PROGRAM Main
VAR
	PowerOn			: bool	:= true;	// initialize on, turn false on second scan
	FirstRun		: BOOL := TRUE;		// initialize on, turn false when system has reached starting postion 

	i						: UINT;				// loop index variable
	Step					: XTSSequence;		// primary sequencer
	stCaGroupRef			: AXES_GROUP_REF;
	fbEnableGroup			: MC_GroupEnable;
	fbAddAxis				: ARRAY[1..GVL.NUM_MOVERS] OF MC_AddAxisToGroup;
	fbRemoveAxisFromGroup	: ARRAY[1..GVL.NUM_MOVERS] OF MC_RemoveAxisFromGroup;
	nAtStart: UINT;
	nToStart: UINT;
	
	allMoversHalted: BOOL;

	
	
	MoversReady: BOOL;
	Started: BOOL;
	Resumed: BOOL;
	bLightCurtainEntered: R_TRIG;
	bLightCurtainExited: F_TRIG;
END_VAR

(* this program handles the main sequencer of this machine *)

// cyclic call to execute fb's for movers, stations, and zones
FOR i := 1 TO GVL.NUM_MOVERS DO
	GVL.Mover[i]();
	GVL.Mover[i].AxisReference.ReadStatus();
	fbRemoveAxisFromGroup[i](AxesGroup		:= stCaGroupRef);
	fbAddAxis[i](AxesGroup		:= stCaGroupRef,
				Axis			:= GVL.Mover[i].AxisReference);
				
	IF GVL.Mover[i].AxisReference.Status.Moving THEN
				allMoversHalted		:= FALSE;
			END_IF
END_FOR
FOR i := 1 TO GVL.NUM_STATIONS DO
	GVL.Station[i]();
END_FOR
FOR i := 1 TO gvl.NUM_ZONES DO
	GVL.Zone[i]();
END_FOR

// check for HMI STOP/PAUSE
IF HMI.Stop THEN
	HMI.Stop	:= FALSE;
	Step		:= XTSSequence.Stop;
ELSIF HMI.Pause THEN
	HMI.Pause	:= FALSE;
	Step		:= XTSSequence.Pause;
END_IF

CASE Step OF

//-----------------------------------------------------------------------------------------------------------------------	
	XTSSequence.Off:
		// state waiting for start command		----	Movers are off
		
		
		
		//COMMIT TEST
		
		Initialize();

			IF HMI.StartOver THEN
				Step		:= XTSSequence.EnableMovers;
				Started := TRUE;
				HMI.StartOver := FALSE;
			END_IF
			
			IF HMI.Resume THEN
				Step			:= XTSSequence.EnableMovers;
				Resumed := TRUE;
				HMI.Resume := FALSE;
			END_IF

//-----------------------------------------------------------------------------------------------------------------------	
	XTSSequence.Pause:
	
	FOR i := 1 TO GVL.NUM_MOVERS  DO
		GVL.Mover[i].toPause := TRUE;
	END_FOR
	
	Started := FALSE;
	Resumed := FALSE;
	Step := XTSSequence.Pausing;
	
//-----------------------------------------------------------------------------------------------------------------------	
	XTSSequence.Pausing:
	
	// Waiting for all to come to a full stop
	allMoversHalted				:= TRUE;
	
	FOR i := 1 TO GVL.NUM_MOVERS DO
		IF GVL.Mover[i].AxisReference.Status.Moving THEN
			allMoversHalted		:= FALSE;
		END_IF
	END_FOR
	
	IF allMoversHalted THEN
		Step		:= XTSSequence.Off;
	END_IF

//-----------------------------------------------------------------------------------------------------------------------	
	XTSSequence.Stop:
	
	FOR i := 1 TO GVL.NUM_MOVERS  DO
		GVL.Mover[i].toStop := TRUE;
	END_FOR
	
	Started := FALSE;
	Resumed := FALSE;
	Step		:= XTSSequence.Stopping;
		
//-----------------------------------------------------------------------------------------------------------------------	
	XTSSequence.Stopping:
		// Waiting for all to come to a full stop
		allMoversHalted				:= TRUE;
	
		FOR i := 1 TO GVL.NUM_MOVERS DO
			IF GVL.Mover[i].AxisReference.Status.Moving THEN
				allMoversHalted		:= FALSE;
			END_IF
		END_FOR
	
	IF allMoversHalted THEN
		Step		:= XTSSequence.RemoveAxes;
	END_IF
	
//-----------------------------------------------------------------------------------------------------------------------	
	XTSSequence.RemoveAxes:
		// remove all axes to collision avoidance group
		// loop through each mover axis and remove CA group
		FOR i:= 1 TO GVL.NUM_MOVERS DO
			fbRemoveAxisFromGroup[i].IdentInGroup := UDINT_TO_IDENTINGROUP(UINT_TO_UDINT(i));
			fbRemoveAxisFromGroup[i].Execute			:= TRUE;
		END_FOR
	
		IF stCaGroupRef.NcToPlc.CA.Common.GroupAxesCount = 0 THEN
			FOR i:= 1 TO GVL.NUM_MOVERS DO
				fbRemoveAxisFromGroup[i].IdentInGroup	:= UDINT_TO_IDENTINGROUP(UINT_TO_UDINT(i));
				fbRemoveAxisFromGroup[i].Execute			:= FALSE;
				MoversReady := FALSE;
		END_FOR
			Step := XTSSequence.DisableMovers;
		END_IF

//-----------------------------------------------------------------------------------------------------------------------	
	XTSSequence.DisableMovers:
	FOR i := 1 TO GVL.NUM_MOVERS  DO
		GVL.Mover[i].toDisable := TRUE;
	END_FOR
	
	Step := XTSSequence.Off;
		
//-----------------------------------------------------------------------------------------------------------------------			
	XTSSequence.EnableMovers:
		// enable all movers
		FOR i := 1 TO GVL.NUM_MOVERS DO
			IF NOT GVL.Mover[i].Enabled THEN
				GVL.Mover[i].Enable	:= TRUE;
			END_IF
		END_FOR
		
		// check for all enabled
		FOR i := 1 TO GVL.NUM_MOVERS DO
			IF NOT GVL.Mover[i].Enabled THEN
				// not enabled, leave for loop
				EXIT;
			END_IF
			// made it this far, all movers are enabled
			IF i = gvl.NUM_MOVERS THEN
				Step	:= XTSSequence.EnableGroup;
			END_IF
		END_FOR
		
//-----------------------------------------------------------------------------------------------------------------------		
	XTSSequence.EnableGroup:
	// enable CA group
	fbEnableGroup.Execute := TRUE;
	// verify group enabled successfully
	IF fbEnableGroup.Done = TRUE THEN
		fbEnableGroup.Execute := FALSE;
		Step := XTSSequence.AddAxes;
	END_IF
		
//-----------------------------------------------------------------------------------------------------------------------		
	XTSSequence.AddAxes:
		// add all axes to collision avoidance group
		// loop through each mover axis and add to CA group
	FOR i:= 1 TO GVL.NUM_MOVERS DO
		fbAddAxis[i].IdentInGroup := UDINT_TO_IDENTINGROUP(UINT_TO_UDINT(i));
		fbAddAxis[i].Execute := TRUE;
	END_FOR
	
	// verify all axes added
	IF stCaGroupRef.NcToPlc.CA.Common.GroupAxesCount = GVL.NUM_MOVERS THEN
		FOR i:= 1 TO GVL.NUM_MOVERS DO
			fbAddAxis[i].IdentInGroup := UDINT_TO_IDENTINGROUP(UINT_TO_UDINT(i));
			fbAddAxis[i].Execute := FALSE;
			MoversReady := TRUE;
			Step	:= XTSSequence.StandBy;
		END_FOR
	END_IF
		
//-----------------------------------------------------------------------------------------------------------------------		
	XTSSequence.StandBy:
	IF Started THEN
		// first time code executes this far (after power on) move to a start position
		Started := FALSE;
		Step	:= XTSSequence.Start;
	ELSIF Resumed THEN
		// any other time code executes here, resume operation where movers left off
		Resumed := FALSE;
		Step	:= XTSSequence.Run;
	END_IF

//-----------------------------------------------------------------------------------------------------------------------		
	XTSSequence.Start:
		// request all movers proceed to starting station
IF HMI.bzone0Stop = FALSE THEN
	FOR i:= 1 TO GVL.NUM_MOVERS DO
		GVL.Mover[i].toStart	:= TRUE;
	END_FOR
	// verify one mover is at start, all others have commands and are at zero speed
	nAtStart	:= 0;
	nToStart	:= 0;
	FOR i:= 1 TO GVL.NUM_MOVERS DO
		IF GVL.Mover[i].Step = MoverSequence.AtStart THEN
			nAtStart	:= nAtStart + 1;
		ELSIF GVL.Mover[i].Step = MoverSequence.MovingToStart THEN
			nToStart	:= nToStart + 1;
		END_IF
	END_FOR
	IF nAtStart = 1 AND nToStart = GVL.NUM_MOVERS - 1 THEN
		Step	:= XTSSequence.Run;
	END_IF
END_IF	
//-----------------------------------------------------------------------------------------------------------------------	
	XTSSequence.Run:
	(*
	FOR i:= 1 TO GVL.NUM_MOVERS DO
			GVL.Mover[i].toNext	:= TRUE;
		END_FOR
	*)
	
	// LOAD TRAY STATION
	IF GVL.Station[1].Step = StationSequence.MoverPresent THEN
		HMI.dsMoverControlFlags.loadTray_Busy := TRUE;
		IF HMI.dsMoverControlFlags.loadTray_Complete THEN			//IF SENSOR IS TRUE PACKAGE IS PRESENT MOVER GOES TO NEXT STATION
			HMI.dsMoverControlFlags.loadTray_Complete := FALSE;
			GVL.Station[1].bMoveToNext := TRUE;
		END_IF
	ELSE
		HMI.dsMoverControlFlags.loadTray_Busy := FALSE;
	END_IF
	
	// LOAD PARTS STATION 1
	IF GVL.Station[2].Step = StationSequence.MoverPresent THEN
		HMI.dsMoverControlFlags.loadArea1_Busy := TRUE;				//SIGNAL TO ROBOT 1 TO LOAD PARTS
		IF HMI.dsMoverControlFlags.loadArea1_Complete THEN			//SIGNAL FROM ROBOT 1 PARTS COMPLETED
			HMI.dsMoverControlFlags.loadArea1_Complete := FALSE;
			GVL.Station[2].bMoveToNext := TRUE;
		END_IF
	ELSE 
		HMI.dsMoverControlFlags.loadArea1_Busy := FALSE;
	END_IF
	
	// LOAD PARTS STATION 2
	IF GVL.Station[3].Step = StationSequence.MoverPresent THEN
		HMI.dsMoverControlFlags.loadArea2_Busy := TRUE;				//SIGNAL TO ROBOT 2 TO LOAD PARTS
		IF HMI.dsMoverControlFlags.loadArea2_Complete THEN			//SIGNAL FROM ROBOT 2 PARTS COMPLETED
			HMI.dsMoverControlFlags.loadArea2_Complete := FALSE;
			GVL.Station[3].bMoveToNext := TRUE;
		END_IF
	ELSE
		HMI.dsMoverControlFlags.loadArea2_Busy := FALSE;	
	END_IF
	
	// LOAD PARTS STATION 3
	IF GVL.Station[4].Step = StationSequence.MoverPresent THEN
		HMI.dsMoverControlFlags.loadArea3_Busy := TRUE;				//SIGNAL TO ROBOT 3 TO LOAD PARTS
		IF HMI.dsMoverControlFlags.loadArea3_Complete THEN			//SIGNAL FROM ROBOT 3 PARTS COMPLETED
			HMI.dsMoverControlFlags.loadArea3_Complete := FALSE;
			GVL.Station[4].bMoveToNext := TRUE;
		END_IF
	ELSE
		HMI.dsMoverControlFlags.loadArea3_Busy := FALSE;
	END_IF

	// LOAD PARTS STATION 4
	IF GVL.Station[5].Step = StationSequence.MoverPresent THEN
		HMI.dsMoverControlFlags.loadArea4_Busy := TRUE;				//SIGNAL TO ROBOT 4 TO LOAD PARTS
		IF HMI.dsMoverControlFlags.loadArea4_Complete THEN			//SIGNAL FROM ROBOT 4 PARTS COMPLETED
			HMI.dsMoverControlFlags.loadArea4_Complete := FALSE;
			GVL.Station[5].bMoveToNext := TRUE;
		END_IF
	ELSE
		HMI.dsMoverControlFlags.loadArea4_Busy := FALSE;	
	END_IF
	
	// UNLOAD PARTS STATION 
	IF GVL.Station[6].Step = StationSequence.MoverPresent THEN
		HMI.dsMoverControlFlags.unloadTray_Busy := TRUE;			//SIGNAL TO ROBOT 5 TO UNLOAD TRAY
		IF HMI.dsMoverControlFlags.unloadTray_Complete THEN			//SIGNAL FROM ROBOT 5 UNLOAD TRAY COMPLETED
			HMI.dsMoverControlFlags.unloadTray_Complete := FALSE;
			IF HMI.bzone0Stop THEN
				GVL.Station[6].bMoveToNext := TRUE;					//Send to Queue Movers Station
			ELSE
				GVL.Station[6].bMoveToStart := TRUE;					//Send to Load Tray Station
			END_IF

		END_IF
	ELSE
		HMI.dsMoverControlFlags.unloadTray_Busy := FALSE;
	END_IF
	
	// Queue Station used only if Operator is in Zone 1
	IF GVL.Station[7].Step = StationSequence.MoverPresent THEN
		IF HMI.bzone0Stop = FALSE THEN			
			GVL.Station[7].bMoveToStart := TRUE;
		END_IF
	END_IF
	
	IF HMI.StartOver THEN
		Started := TRUE;
		HMI.StartOver := FALSE;
		Step :=	XTSSequence.Standby;
		
	END_IF
	
END_CASE

fbEnableGroup(AxesGroup	:= stCaGroupRef);
LightCurtainCheck();

METHOD Initialize : BOOL
VAR_INPUT
END_VAR
// set values of function blocks
	GVL.Station[1].Position		:= 0.0;
	GVL.Station[2].Position		:= 750.0;
	GVL.Station[3].Position		:= 1500.0;
	GVL.Station[4].Position		:= 2250.0;
	GVL.Station[5].Position		:= 3000.0;
	GVL.Station[6].Position		:= 3600.0;
	GVL.Station[7].Position		:= 4250.0;
	GVL.Station[8].Position		:= 4490.0;
END_METHOD

ACTION LightCurtainCheck:
// ZONE 0  OPERATER LOADING
bLightCurtainEntered(CLK:=HMI.bzone0Stop);
bLightCurtainExited(CLK:=HMI.bzone0Stop);
	IF bLightCurtainEntered.Q THEN
		FOR i:= 1 TO GVL.NUM_MOVERS DO	
			IF GVL.Mover[i].Position >= 4500.0 OR GVL.Mover[i].Position <= 500.0 THEN
			GVL.Mover[i].toPause	:= TRUE;
			GVL.Mover[i].toNext		:= FALSE;
			GVL.Mover[i].toStart	:= FALSE;
			END_IF
		END_FOR
	END_IF
	IF bLightCurtainExited.Q THEN
		FOR i:= 1 TO GVL.NUM_MOVERS DO	
			IF GVL.Mover[i].Position > 4500.0 THEN
				GVL.Mover[i].toStart	:= TRUE;
			END_IF
		END_FOR
	END_IF
END_ACTION

END_PROGRAM

(* stored: Version 1.1.0.1, ProductVersion 3.1.4026.8
   POU Main: Id {99d93c32-af77-0b47-2160-e8a9eed47eae}, SpecialFunc None
   Method Initialize: Id {4ea4d127-ec11-0953-31c9-c3462af2cac5}
   Action LightCurtainCheck: Id {c8440321-cf39-0d36-2897-bf963226c8e3} *)
